KUKA KRL data list: ps_a_etb_res_c02.dat

&ACCESS RVO1
&REL 341
&COMMENT Solda Atego ETB
&PARAM DISKPATH = KRC:\R1\Program\OLP
DEFDAT  ps_a_etb_res_c02
;FOLD EXTERNAL DECLARATIONS;%{PE}%MKUKATPBASIS,%CEXT,%VCOMMON,%P
;FOLD GRIPPERTECH EXT
EXT  H50 (INT  :IN,INT  :IN,INT  :IN,GRP_TYP  :IN )
;ENDFOLD (GRIPPERTECH EXT)
;FOLD SPOTTECH EXT
EXT  USERSPOT (S_COMMAND  :IN,SPOT_TYPE  :IN )
;ENDFOLD (SPOTTECH EXT)
;FOLD BASISTECH EXT;%{PE}%MKUKATPBASIS,%CEXT,%VEXT,%P
EXT  BAS (BAS_COMMAND  :IN,REAL  :IN )
DECL INT SUCCESS
;ENDFOLD (BASISTECH EXT)
;FOLD USER EXT;%{E}%MKUKATPUSER,%CEXT,%VEXT,%P
;Make your modifications here

;ENDFOLD (USER EXT)
;ENDFOLD (EXTERNAL DECLARATIONS)
DECL FDAT Fl015={TOOL_NO 3,BASE_NO 3,IPO_FRAME #BASE,POINT2[] " "}
DECL E6POS Xl015={X 31.0238705,Y -594.734375,Z 749.761108,A -124.005302,B 73.4685669,C -126.8536,S 18,T 35,E1 0.0,E2 0.0,E3 0.0,E4 0.0,E5 0.0,E6 0.0}
DECL LDAT LL_OLP3={VEL 2.0,ACC 100.0,APO_DIST 0.0,APO_FAC 0.0,ORI_TYP #VAR,CIRC_TYP #BASE,JERK_FAC 50.0}
DECL FDAT Fl020={TOOL_NO 3,BASE_NO 3,IPO_FRAME #BASE,POINT2[] " "}
DECL E6POS Xl020={X 52.5596504,Y -663.980286,Z 782.928284,A -123.990501,B 73.4740219,C -126.844803,S 18,T 35,E1 0.0,E2 0.0,E3 0.0,E4 0.0,E5 0.0,E6 0.0}
DECL LDAT LL_OLP4={VEL 2.0,ACC 100.0,APO_DIST 150.0,APO_FAC 0.0,ORI_TYP #VAR,CIRC_TYP #BASE,JERK_FAC 50.0}
DECL FDAT Fl025={TOOL_NO 3,BASE_NO 3,IPO_FRAME #BASE,POINT2[] " "}
DECL E6POS Xl025={X 114.589798,Y -708.233398,Z 735.784912,A -94.4452896,B 74.9285278,C -94.8186569,S 18,T 35,E1 0.0,E2 0.0,E3 0.0,E4 0.0,E5 0.0,E6 0.0}
DECL LDAT LL_OLP5={VEL 2.0,ACC 100.0,APO_DIST 150.0,APO_FAC 0.0,ORI_TYP #VAR,CIRC_TYP #BASE,JERK_FAC 50.0}
DECL FDAT Fl030={TOOL_NO 3,BASE_NO 3,IPO_FRAME #BASE,POINT2[] " "}
DECL E6POS Xl030={X 274.340912,Y -703.442017,Z 641.453125,A -54.7125397,B 69.4866562,C -51.1110687,S 18,T 35,E1 0.0,E2 0.0,E3 0.0,E4 0.0,E5 0.0,E6 0.0}
DECL LDAT LL_OLP6={VEL 2.0,ACC 100.0,APO_DIST 150.0,APO_FAC 0.0,ORI_TYP #VAR,CIRC_TYP #BASE,JERK_FAC 50.0}
DECL FDAT Fl035={TOOL_NO 3,BASE_NO 3,IPO_FRAME #BASE,POINT2[] " "}
DECL E6POS Xl035={X 587.583008,Y -653.065002,Z 418.535004,A -24.4300995,B 45.0119019,C -12.2528,S 2,T 35}
DECL LDAT LL_OLP7={VEL 2.0,ACC 100.0,APO_DIST 150.0,APO_FAC 0.0,ORI_TYP #VAR,CIRC_TYP #BASE,JERK_FAC 50.0}
DECL FDAT Fl040={TOOL_NO 3,BASE_NO 3,IPO_FRAME #BASE,POINT2[] " "}
DECL E6POS Xl040={X 713.926392,Y -668.47052,Z 338.3591,A -21.6110992,B 32.5932884,C -7.47571993,S 18,T 35,E1 0.0,E2 0.0,E3 0.0,E4 0.0,E5 0.0,E6 0.0}
DECL LDAT LL_OLP8={VEL 2.0,ACC 100.0,APO_DIST 150.0,APO_FAC 0.0,ORI_TYP #VAR,CIRC_TYP #BASE,JERK_FAC 50.0}
DECL FDAT Fl045={TOOL_NO 3,BASE_NO 3,IPO_FRAME #BASE,POINT2[] " "}
DECL E6POS Xl045={X 765.193115,Y -1115.46997,Z 133.110596,A -16.9657192,B 14.9491901,C -20.2578106,S 18,T 3,E1 0.0,E2 0.0,E3 0.0,E4 0.0,E5 0.0,E6 0.0}
DECL LDAT LL_OLP9={VEL 2.0,ACC 100.0,APO_DIST 150.0,APO_FAC 0.0,ORI_TYP #VAR,CIRC_TYP #BASE,JERK_FAC 50.0}
DECL FDAT Fl050={TOOL_NO 3,BASE_NO 3,IPO_FRAME #BASE,POINT2[] " "}
DECL E6POS Xl050={X 746.955017,Y -2151.34399,Z 121.584,A -16.3197002,B 12.0216999,C -22.6774998,S 2,T 3}
DECL FDAT Fl055={TOOL_NO 3,BASE_NO 3,IPO_FRAME #BASE,POINT2[] " "}
DECL E6POS Xl055={X 1024.95605,Y -2151.34399,Z 535.583008,A 28.6604996,B 24.3521996,C -7.86679983,S 2,T 3}
DECL FDAT Fl060={TOOL_NO 3,BASE_NO 3,IPO_FRAME #BASE,POINT2[] " "}
DECL PDAT PP_OLP2={VEL 100.0,ACC 100.0,APO_DIST 100.0,APO_MODE #CDIS}
DECL E6POS Xl060={X 1158.77795,Y -1627.54797,Z 929.039001,A 43.2759018,B -40.0696983,C 26.0069008,S 6,T 19}
DECL FDAT Fl065={TOOL_NO 3,BASE_NO 3,IPO_FRAME #BASE,POINT2[] " "}
DECL PDAT PP_OLP3={VEL 100.0,ACC 100.0,APO_DIST 30.0,APO_MODE #CDIS}
DECL E6POS Xl065={X 868.09668,Y -1244.59497,Z 1101.58606,A 29.2385902,B -63.5374794,C 57.4689713,S 22,T 19,E1 0.0,E2 0.0,E3 0.0,E4 0.0,E5 0.0,E6 0.0}
DECL FDAT Fl070={TOOL_NO 3,BASE_NO 3,IPO_FRAME #BASE,POINT2[] " "}
DECL PDAT PP_OLP4={VEL 100.0,ACC 100.0,APO_DIST 30.0,APO_MODE #CDIS}
DECL E6POS Xl070={X 814.102905,Y -929.709717,Z 1165.05896,A 29.5652695,B -64.2360001,C 60.087719,S 22,T 19,E1 0.0,E2 0.0,E3 0.0,E4 0.0,E5 0.0,E6 0.0}
DECL E6POS XSWP_60_7787={X 556.251099,Y -975.593323,Z 1302.83704,A 143.936295,B -83.3156891,C -51.7027016,S 18,T 43,E1 0.0,E2 0.0,E3 0.0,E4 0.0,E5 0.0,E6 0.0}
DECL FDAT FSWP_60_7787={TOOL_NO 3,BASE_NO 3,IPO_FRAME #BASE,POINT2[] " "}
DECL LDAT LL_OLP12={VEL 2.0,ACC 100.0,APO_DIST 0.0,APO_FAC 0.0,ORI_TYP #VAR,CIRC_TYP #BASE,JERK_FAC 50.0}
DECL E6POS XSWP_60_7789={X 584.018677,Y -975.191223,Z 1304.28101,A 144.007706,B -83.3220673,C -54.6376801,S 18,T 43,E1 0.0,E2 0.0,E3 0.0,E4 0.0,E5 0.0,E6 0.0}
DECL FDAT FSWP_60_7789={TOOL_NO 3,BASE_NO 3,IPO_FRAME #BASE,POINT2[] " "}
DECL LDAT LL_OLP13={VEL 2.0,ACC 100.0,APO_DIST 0.0,APO_FAC 0.0,ORI_TYP #VAR,CIRC_TYP #BASE,JERK_FAC 50.0}
DECL E6POS XSWP_60_7791={X 613.247986,Y -978.535706,Z 1306.79395,A 144.016205,B -83.3237762,C -54.6469498,S 22,T 19,E1 0.0,E2 0.0,E3 0.0,E4 0.0,E5 0.0,E6 0.0}
DECL FDAT FSWP_60_7791={TOOL_NO 3,BASE_NO 3,IPO_FRAME #BASE,POINT2[] " "}
DECL LDAT LL_OLP14={VEL 2.0,ACC 100.0,APO_DIST 0.0,APO_FAC 0.0,ORI_TYP #VAR,CIRC_TYP #BASE,JERK_FAC 50.0}
DECL FDAT Fl075={TOOL_NO 3,BASE_NO 3,IPO_FRAME #BASE,POINT2[] " "}
DECL E6POS Xl075={X 647.49408,Y -968.108398,Z 1301.578,A 26.10993,B -81.5293198,C 62.8230019,S 22,T 19,E1 0.0,E2 0.0,E3 0.0,E4 0.0,E5 0.0,E6 0.0}
DECL LDAT LL_OLP15={VEL 2.0,ACC 100.0,APO_DIST 10.0,APO_FAC 0.0,ORI_TYP #VAR,CIRC_TYP #BASE,JERK_FAC 50.0}
DECL E6POS XSWP_60_7795={X 702.531372,Y -979.488403,Z 1310.90405,A 26.1140499,B -81.5290985,C 62.8173103,S 22,T 19,E1 0.0,E2 0.0,E3 0.0,E4 0.0,E5 0.0,E6 0.0}
DECL FDAT FSWP_60_7795={TOOL_NO 3,BASE_NO 3,IPO_FRAME #BASE,POINT2[] " "}
DECL LDAT LL_OLP16={VEL 2.0,ACC 100.0,APO_DIST 0.0,APO_FAC 0.0,ORI_TYP #VAR,CIRC_TYP #BASE,JERK_FAC 50.0}
DECL E6POS XSWP_60_7797={X 744.206726,Y -979.352295,Z 1312.43701,A 26.1139603,B -81.5292435,C 62.8172798,S 22,T 19,E1 0.0,E2 0.0,E3 0.0,E4 0.0,E5 0.0,E6 0.0}
DECL FDAT FSWP_60_7797={TOOL_NO 3,BASE_NO 3,IPO_FRAME #BASE,POINT2[] " "}
DECL LDAT LL_OLP17={VEL 2.0,ACC 100.0,APO_DIST 0.0,APO_FAC 0.0,ORI_TYP #VAR,CIRC_TYP #BASE,JERK_FAC 50.0}
DECL E6POS XSWP_60_7799={X 790.615112,Y -980.393005,Z 1313.89502,A 26.1141491,B -81.5294495,C 62.8168793,S 22,T 19,E1 0.0,E2 0.0,E3 0.0,E4 0.0,E5 0.0,E6 0.0}
DECL FDAT FSWP_60_7799={TOOL_NO 3,BASE_NO 3,IPO_FRAME #BASE,POINT2[] " "}
DECL LDAT LL_OLP18={VEL 2.0,ACC 100.0,APO_DIST 0.0,APO_FAC 0.0,ORI_TYP #VAR,CIRC_TYP #BASE,JERK_FAC 50.0}
DECL E6POS XSWP_60_7801={X 838.112976,Y -981.874023,Z 1316.401,A 26.1212902,B -81.5292511,C 62.8090897,S 22,T 19,E1 0.0,E2 0.0,E3 0.0,E4 0.0,E5 0.0,E6 0.0}
DECL FDAT FSWP_60_7801={TOOL_NO 3,BASE_NO 3,IPO_FRAME #BASE,POINT2[] " "}
DECL LDAT LL_OLP19={VEL 2.0,ACC 100.0,APO_DIST 0.0,APO_FAC 0.0,ORI_TYP #VAR,CIRC_TYP #BASE,JERK_FAC 50.0}
DECL E6POS XSWP_60_7803={X 879.085815,Y -982.434204,Z 1317.19104,A 26.1254692,B -81.5289612,C 62.8045807,S 22,T 19,E1 0.0,E2 0.0,E3 0.0,E4 0.0,E5 0.0,E6 0.0}
DECL FDAT FSWP_60_7803={TOOL_NO 3,BASE_NO 3,IPO_FRAME #BASE,POINT2[] " "}
DECL LDAT LL_OLP20={VEL 2.0,ACC 100.0,APO_DIST 0.0,APO_FAC 0.0,ORI_TYP #VAR,CIRC_TYP #BASE,JERK_FAC 50.0}
DECL E6POS XSWP_60_7807={X 972.588501,Y -983.796387,Z 1320.14001,A 26.1272507,B -81.5321884,C 62.805069,S 22,T 19,E1 0.0,E2 0.0,E3 0.0,E4 0.0,E5 0.0,E6 0.0}
DECL FDAT FSWP_60_7807={TOOL_NO 3,BASE_NO 3,IPO_FRAME #BASE,POINT2[] " "}
DECL LDAT LL_OLP21={VEL 2.0,ACC 100.0,APO_DIST 0.0,APO_FAC 0.0,ORI_TYP #VAR,CIRC_TYP #BASE,JERK_FAC 50.0}
DECL E6POS XSWP_60_7809={X 1019.99597,Y -984.109985,Z 1320.86499,A 26.1021805,B -81.5284271,C 62.8301506,S 22,T 19,E1 0.0,E2 0.0,E3 0.0,E4 0.0,E5 0.0,E6 0.0}
DECL FDAT FSWP_60_7809={TOOL_NO 3,BASE_NO 3,IPO_FRAME #BASE,POINT2[] " "}
DECL LDAT LL_OLP22={VEL 2.0,ACC 100.0,APO_DIST 0.0,APO_FAC 0.0,ORI_TYP #VAR,CIRC_TYP #BASE,JERK_FAC 50.0}
DECL E6POS XSWP_60_7811={X 1062.02405,Y -985.307312,Z 1321.88196,A 26.1204891,B -81.530159,C 62.8099213,S 22,T 19,E1 0.0,E2 0.0,E3 0.0,E4 0.0,E5 0.0,E6 0.0}
DECL FDAT FSWP_60_7811={TOOL_NO 3,BASE_NO 3,IPO_FRAME #BASE,POINT2[] " "}
DECL LDAT LL_OLP23={VEL 2.0,ACC 100.0,APO_DIST 0.0,APO_FAC 0.0,ORI_TYP #VAR,CIRC_TYP #BASE,JERK_FAC 50.0}
DECL E6POS XSWP_60_7813={X 1102.52795,Y -985.327515,Z 1323.27405,A 26.1103802,B -81.5287933,C 62.8201218,S 22,T 19,E1 0.0,E2 0.0,E3 0.0,E4 0.0,E5 0.0,E6 0.0}
DECL FDAT FSWP_60_7813={TOOL_NO 3,BASE_NO 3,IPO_FRAME #BASE,POINT2[] " "}
DECL LDAT LL_OLP24={VEL 2.0,ACC 100.0,APO_DIST 0.0,APO_FAC 0.0,ORI_TYP #VAR,CIRC_TYP #BASE,JERK_FAC 50.0}
DECL E6POS XSWP_60_7815={X 1147.90198,Y -985.572815,Z 1324.37402,A 26.1104202,B -81.528923,C 62.8199615,S 22,T 19,E1 0.0,E2 0.0,E3 0.0,E4 0.0,E5 0.0,E6 0.0}
DECL FDAT FSWP_60_7815={TOOL_NO 3,BASE_NO 3,IPO_FRAME #BASE,POINT2[] " "}
DECL LDAT LL_OLP25={VEL 2.0,ACC 100.0,APO_DIST 0.0,APO_FAC 0.0,ORI_TYP #VAR,CIRC_TYP #BASE,JERK_FAC 50.0}
DECL FDAT Fl080={TOOL_NO 3,BASE_NO 3,IPO_FRAME #BASE,POINT2[] " "}
DECL E6POS Xl080={X 1163.40503,Y -974.013977,Z 1320.32605,A 13.9886799,B -81.9076538,C 74.8192825,S 22,T 19,E1 0.0,E2 0.0,E3 0.0,E4 0.0,E5 0.0,E6 0.0}
DECL LDAT LL_OLP26={VEL 2.0,ACC 100.0,APO_DIST 150.0,APO_FAC 0.0,ORI_TYP #VAR,CIRC_TYP #BASE,JERK_FAC 50.0}
DECL FDAT Fl085={TOOL_NO 3,BASE_NO 3,IPO_FRAME #BASE,POINT2[] " "}
DECL E6POS Xl085={X 1163.94604,Y -969.89032,Z 1259.79297,A 17.7539597,B -81.8335037,C 71.0904465,S 22,T 19,E1 0.0,E2 0.0,E3 0.0,E4 0.0,E5 0.0,E6 0.0}
DECL LDAT LL_OLP27={VEL 2.0,ACC 100.0,APO_DIST 150.0,APO_FAC 0.0,ORI_TYP #VAR,CIRC_TYP #BASE,JERK_FAC 50.0}
DECL FDAT Fl090={TOOL_NO 3,BASE_NO 3,IPO_FRAME #BASE,POINT2[] " "}
DECL E6POS Xl090={X 983.369995,Y -1478.85596,Z 590.278015,A 179.957108,B -45.9999008,C -90.0,S 6,T 19}
DECL LDAT LL_OLP28={VEL 2.0,ACC 100.0,APO_DIST 150.0,APO_FAC 0.0,ORI_TYP #VAR,CIRC_TYP #BASE,JERK_FAC 50.0}
DECL FDAT Fl100={TOOL_NO 3,BASE_NO 3,IPO_FRAME #BASE,POINT2[] " "}
DECL E6POS Xl100={X 1306.58801,Y -1016.62402,Z 103.935699,A 179.322601,B -25.2803707,C -90.9719391,S 22,T 19,E1 0.0,E2 0.0,E3 0.0,E4 0.0,E5 0.0,E6 0.0}
DECL LDAT LL_OLP30={VEL 2.0,ACC 100.0,APO_DIST 0.0,APO_FAC 0.0,ORI_TYP #VAR,CIRC_TYP #BASE,JERK_FAC 50.0}
DECL FDAT FSWP_60_7487={TOOL_NO 3,BASE_NO 3,IPO_FRAME #BASE,POINT2[] " "}
DECL E6POS XSWP_60_7487={X 1306.44397,Y -1021.547,Z 118.262802,A 179.322403,B -25.28022,C -90.9719391,S 18,T 43,E1 0.0,E2 0.0,E3 0.0,E4 0.0,E5 0.0,E6 0.0}
DECL LDAT LL_OLP31={VEL 2.0,ACC 100.0,APO_DIST 0.0,APO_FAC 0.0,ORI_TYP #VAR,CIRC_TYP #BASE,JERK_FAC 50.0}
DECL FDAT FSWP_60_7489={TOOL_NO 3,BASE_NO 3,IPO_FRAME #BASE,POINT2[] " "}
DECL E6POS XSWP_60_7489={X 1339.98206,Y -1023.56598,Z 120.081001,A 179.952698,B -20.9994793,C -93.3431702,S 18,T 43,E1 0.0,E2 0.0,E3 0.0,E4 0.0,E5 0.0,E6 0.0}
DECL LDAT LL_OLP32={VEL 2.0,ACC 100.0,APO_DIST 0.0,APO_FAC 0.0,ORI_TYP #VAR,CIRC_TYP #BASE,JERK_FAC 50.0}
DECL FDAT FSWP_60_7491={TOOL_NO 3,BASE_NO 3,IPO_FRAME #BASE,POINT2[] " "}
DECL E6POS XSWP_60_7491={X 1370.55298,Y -1021.91803,Z 121.484901,A -179.790604,B -20.8528404,C -93.2146988,S 18,T 43,E1 0.0,E2 0.0,E3 0.0,E4 0.0,E5 0.0,E6 0.0}
DECL LDAT LL_OLP33={VEL 2.0,ACC 100.0,APO_DIST 0.0,APO_FAC 0.0,ORI_TYP #VAR,CIRC_TYP #BASE,JERK_FAC 50.0}
DECL FDAT Fl105={TOOL_NO 3,BASE_NO 3,IPO_FRAME #BASE,POINT2[] " "}
DECL E6POS Xl105={X 1373.94495,Y -1013.10602,Z 88.1965637,A 179.956894,B -18.0000401,C -89.9994507,S 22,T 19,E1 0.0,E2 0.0,E3 0.0,E4 0.0,E5 0.0,E6 0.0}
DECL LDAT LL_OLP34={VEL 2.0,ACC 100.0,APO_DIST 0.0,APO_FAC 0.0,ORI_TYP #VAR,CIRC_TYP #BASE,JERK_FAC 50.0}
DECL FDAT Fl110={TOOL_NO 3,BASE_NO 3,IPO_FRAME #BASE,POINT2[] " "}
DECL E6POS Xl110={X 1469.69604,Y -999.753174,Z 86.6159668,A 179.956894,B -19.0000801,C -89.9993668,S 22,T 19,E1 0.0,E2 0.0,E3 0.0,E4 0.0,E5 0.0,E6 0.0}
DECL LDAT LL_OLP35={VEL 2.0,ACC 100.0,APO_DIST 0.0,APO_FAC 0.0,ORI_TYP #VAR,CIRC_TYP #BASE,JERK_FAC 50.0}
DECL FDAT FSWP_60_7495={TOOL_NO 3,BASE_NO 3,IPO_FRAME #BASE,POINT2[] " "}
DECL E6POS XSWP_60_7495={X 1442.27197,Y -1019.48102,Z 122.377296,A 179.957199,B -20.9995899,C -93.1918564,S 22,T 19,E1 0.0,E2 0.0,E3 0.0,E4 0.0,E5 0.0,E6 0.0}
DECL LDAT LL_OLP36={VEL 2.0,ACC 100.0,APO_DIST 0.0,APO_FAC 0.0,ORI_TYP #VAR,CIRC_TYP #BASE,JERK_FAC 50.0}
DECL FDAT FSWP_60_7497={TOOL_NO 3,BASE_NO 3,IPO_FRAME #BASE,POINT2[] " "}
DECL E6POS XSWP_60_7497={X 1479.71106,Y -1018.96399,Z 124.096703,A -179.6689,B -20.9927502,C -93.8000717,S 18,T 43,E1 0.0,E2 0.0,E3 0.0,E4 0.0,E5 0.0,E6 0.0}
DECL LDAT LL_OLP37={VEL 2.0,ACC 100.0,APO_DIST 0.0,APO_FAC 0.0,ORI_TYP #VAR,CIRC_TYP #BASE,JERK_FAC 50.0}
DECL FDAT FSWP_60_7499={TOOL_NO 3,BASE_NO 3,IPO_FRAME #BASE,POINT2[] " "}
DECL E6POS XSWP_60_7499={X 1519.71802,Y -1018.96802,Z 124.852798,A -179.660904,B -20.9865093,C -93.8057938,S 18,T 43,E1 0.0,E2 0.0,E3 0.0,E4 0.0,E5 0.0,E6 0.0}
DECL LDAT LL_OLP38={VEL 2.0,ACC 100.0,APO_DIST 0.0,APO_FAC 0.0,ORI_TYP #VAR,CIRC_TYP #BASE,JERK_FAC 50.0}
DECL FDAT Fl115={TOOL_NO 3,BASE_NO 3,IPO_FRAME #BASE,POINT2[] " "}
DECL E6POS Xl115={X 1563.23596,Y -1006.01099,Z 70.940239,A 179.949402,B -20.9986,C -89.9980469,S 22,T 19,E1 0.0,E2 0.0,E3 0.0,E4 0.0,E5 0.0,E6 0.0}
DECL LDAT LL_OLP39={VEL 2.0,ACC 100.0,APO_DIST 150.0,APO_FAC 0.0,ORI_TYP #VAR,CIRC_TYP #BASE,JERK_FAC 50.0}
DECL FDAT Fl120={TOOL_NO 3,BASE_NO 3,IPO_FRAME #BASE,POINT2[] " "}
DECL E6POS Xl120={X 1563.09998,Y -1231.07898,Z 75.473999,A 179.957108,B -20.9999008,C -90.0,S 6,T 19}
DECL LDAT LL_OLP40={VEL 2.0,ACC 100.0,APO_DIST 150.0,APO_FAC 0.0,ORI_TYP #VAR,CIRC_TYP #BASE,JERK_FAC 50.0}
DECL FDAT Fl125={TOOL_NO 3,BASE_NO 3,IPO_FRAME #BASE,POINT2[] " "}
DECL E6POS Xl125={X 1667.94995,Y -1726.27698,Z 177.965393,A 179.960098,B -45.9984512,C -90.0082397,S 22,T 19,E1 0.0,E2 0.0,E3 0.0,E4 0.0,E5 0.0,E6 0.0}
DECL BASIS_SUGG_T LAST_BASIS={POINT1[] "P16                     ",POINT2[] "P16                     ",CP_PARAMS[] "CPDAT0                  ",PTP_PARAMS[] "PDAT17                  ",CONT[] "C_DIS                   ",CP_VEL[] "2                       ",PTP_VEL[] "100                     ",SYNC_PARAMS[] "SYNCDAT                 ",SPL_NAME[] "S0                      "}
DECL PDAT PP_OLP6={VEL 100.0,ACC 100.0,APO_DIST 0.0}
DECL E6POS Xl006={X 746.955017,Y -2151.34399,Z 121.584,A -16.3197002,B 12.0216999,C -22.6774998,S 2,T 3}
DECL FDAT Fl006={TOOL_NO 3,BASE_NO 3,IPO_FRAME #BASE,POINT2[] " "}
DECL LDAT LL_OLP42={VEL 2.0,ACC 100.0,APO_DIST 30.0,APO_FAC 0.0,ORI_TYP #VAR,CIRC_TYP #BASE,JERK_FAC 50.0}
DECL E6POS Xl011={X 745.054077,Y -1210.42102,Z 45.7849503,A -16.3183804,B 12.0204601,C -22.6786194,S 18,T 3,E1 0.0,E2 0.0,E3 0.0,E4 0.0,E5 0.0,E6 0.0}
DECL FDAT Fl011={TOOL_NO 3,BASE_NO 3,IPO_FRAME #BASE,POINT2[] " "}
DECL E6POS Xl016={X 960.239685,Y -695.417419,Z 224.849792,A -18.2002106,B 11.2452402,C -1.07748699,S 18,T 3,E1 0.0,E2 0.0,E3 0.0,E4 0.0,E5 0.0,E6 0.0}
DECL FDAT Fl016={TOOL_NO 3,BASE_NO 3,IPO_FRAME #BASE,POINT2[] " "}
DECL LDAT LL_OLP44={VEL 2.0,ACC 100.0,APO_DIST 10.0,APO_FAC 0.0,ORI_TYP #VAR,CIRC_TYP #BASE,JERK_FAC 50.0}
DECL E6POS Xl021={X 587.583008,Y -653.065002,Z 418.535004,A -24.4300995,B 45.0119019,C -12.2528,S 2,T 35}
DECL FDAT Fl021={TOOL_NO 3,BASE_NO 3,IPO_FRAME #BASE,POINT2[] " "}
DECL LDAT LL_OLP45={VEL 2.0,ACC 100.0,APO_DIST 10.0,APO_FAC 0.0,ORI_TYP #VAR,CIRC_TYP #BASE,JERK_FAC 50.0}
DECL E6POS Xl026={X 343.014008,Y -642.028076,Z 721.553772,A -44.0348091,B 69.0998383,C -36.2288399,S 18,T 35,E1 0.0,E2 0.0,E3 0.0,E4 0.0,E5 0.0,E6 0.0}
DECL FDAT Fl026={TOOL_NO 3,BASE_NO 3,IPO_FRAME #BASE,POINT2[] " "}
DECL LDAT LL_OLP46={VEL 2.0,ACC 100.0,APO_DIST 10.0,APO_FAC 0.0,ORI_TYP #VAR,CIRC_TYP #BASE,JERK_FAC 50.0}
DECL E6POS Xl031={X 328.106598,Y -647.627686,Z 744.279175,A -69.6208572,B 74.6609573,C -62.4694595,S 18,T 35,E1 0.0,E2 0.0,E3 0.0,E4 0.0,E5 0.0,E6 0.0}
DECL FDAT Fl031={TOOL_NO 3,BASE_NO 3,IPO_FRAME #BASE,POINT2[] " "}
DECL LDAT LL_OLP47={VEL 2.0,ACC 100.0,APO_DIST 10.0,APO_FAC 0.0,ORI_TYP #VAR,CIRC_TYP #BASE,JERK_FAC 50.0}
DECL E6POS Xl036={X 129.093597,Y -809.958801,Z 712.43811,A -122.0411,B 73.8237534,C -124.462097,S 18,T 35,E1 0.0,E2 0.0,E3 0.0,E4 0.0,E5 0.0,E6 0.0}
DECL FDAT Fl036={TOOL_NO 3,BASE_NO 3,IPO_FRAME #BASE,POINT2[] " "}
DECL LDAT LL_OLP48={VEL 2.0,ACC 100.0,APO_DIST 10.0,APO_FAC 0.0,ORI_TYP #VAR,CIRC_TYP #BASE,JERK_FAC 50.0}
DECL E6POS Xl041={X 111.864998,Y -869.716003,Z 602.434021,A -124.114799,B 73.5134964,C -126.966202,S 2,T 35}
DECL FDAT Fl041={TOOL_NO 3,BASE_NO 3,IPO_FRAME #BASE,POINT2[] " "}
DECL LDAT LL_OLP49={VEL 2.0,ACC 100.0,APO_DIST 0.0,APO_FAC 0.0,ORI_TYP #VAR,CIRC_TYP #BASE,JERK_FAC 50.0}
DECL E6POS XSWP_60_7909={X 133.370605,Y -867.391907,Z 600.803284,A -109.557999,B 75.6781464,C -117.705002,S 18,T 35,E1 0.0,E2 0.0,E3 0.0,E4 0.0,E5 0.0,E6 0.0}
DECL FDAT FSWP_60_7909={TOOL_NO 3,BASE_NO 3,IPO_FRAME #BASE,POINT2[] " "}
DECL E6POS XSWP_60_7907={X 129.188995,Y -831.960022,Z 602.795776,A -109.579597,B 75.6635437,C -112.607803,S 18,T 35,E1 0.0,E2 0.0,E3 0.0,E4 0.0,E5 0.0,E6 0.0}
DECL FDAT FSWP_60_7907={TOOL_NO 3,BASE_NO 3,IPO_FRAME #BASE,POINT2[] " ",TQ_STATE FALSE}
DECL LDAT LL_OLP51={VEL 2.0,ACC 100.0,APO_DIST 0.0,APO_FAC 0.0,ORI_TYP #VAR,CIRC_TYP #BASE,JERK_FAC 50.0}
DECL E6POS XSWP_60_7905={X 118.431503,Y -758.19519,Z 600.044189,A -94.7613678,B 76.664772,C -98.2709122,S 18,T 35,E1 0.0,E2 0.0,E3 0.0,E4 0.0,E5 0.0,E6 0.0}
DECL FDAT FSWP_60_7905={TOOL_NO 3,BASE_NO 3,IPO_FRAME #BASE,POINT2[] " "}
DECL LDAT LL_OLP52={VEL 2.0,ACC 100.0,APO_DIST 0.0,APO_FAC 0.0,ORI_TYP #VAR,CIRC_TYP #BASE,JERK_FAC 50.0}
DECL E6POS XSWP_60_7903={X 114.063904,Y -728.930908,Z 599.57019,A -101.589203,B 80.7481232,C -104.514198,S 18,T 35,E1 0.0,E2 0.0,E3 0.0,E4 0.0,E5 0.0,E6 0.0}
DECL FDAT FSWP_60_7903={TOOL_NO 3,BASE_NO 3,IPO_FRAME #BASE,POINT2[] " "}
DECL LDAT LL_OLP53={VEL 2.0,ACC 100.0,APO_DIST 0.0,APO_FAC 0.0,ORI_TYP #VAR,CIRC_TYP #BASE,JERK_FAC 50.0}
DECL E6POS XSWP_60_7901={X 112.070602,Y -698.476318,Z 599.263123,A -103.006798,B 80.6964798,C -105.953697,S 18,T 35,E1 0.0,E2 0.0,E3 0.0,E4 0.0,E5 0.0,E6 0.0}
DECL FDAT FSWP_60_7901={TOOL_NO 3,BASE_NO 3,IPO_FRAME #BASE,POINT2[] " "}
DECL LDAT LL_OLP54={VEL 2.0,ACC 100.0,APO_DIST 0.0,APO_FAC 0.0,ORI_TYP #VAR,CIRC_TYP #BASE,JERK_FAC 50.0}
DECL E6POS XSWP_60_7329={X 100.614502,Y -668.871277,Z 599.434021,A -105.788803,B 80.5839996,C -108.767899,S 18,T 35,E1 0.0,E2 0.0,E3 0.0,E4 0.0,E5 0.0,E6 0.0}
DECL FDAT FSWP_60_7329={TOOL_NO 3,BASE_NO 3,IPO_FRAME #BASE,POINT2[] " "}
DECL LDAT LL_OLP55={VEL 2.0,ACC 100.0,APO_DIST 0.0,APO_FAC 0.0,ORI_TYP #VAR,CIRC_TYP #BASE,JERK_FAC 50.0}
DECL E6POS XSWP_60_7893={X 98.5761185,Y -581.989014,Z 599.465881,A -106.232101,B 80.5538635,C -106.072998,S 18,T 35,E1 0.0,E2 0.0,E3 0.0,E4 0.0,E5 0.0,E6 0.0}
DECL FDAT FSWP_60_7893={TOOL_NO 3,BASE_NO 3,IPO_FRAME #BASE,POINT2[] " "}
DECL LDAT LL_OLP56={VEL 2.0,ACC 100.0,APO_DIST 0.0,APO_FAC 0.0,ORI_TYP #VAR,CIRC_TYP #BASE,JERK_FAC 50.0}
DECL E6POS XSWP_60_7891={X 101.4776,Y -547.356323,Z 601.088318,A -147.087204,B 85.1514587,C -145.4216,S 18,T 35,E1 0.0,E2 0.0,E3 0.0,E4 0.0,E5 0.0,E6 0.0}
DECL FDAT FSWP_60_7891={TOOL_NO 3,BASE_NO 3,IPO_FRAME #BASE,POINT2[] " "}
DECL LDAT LL_OLP57={VEL 2.0,ACC 100.0,APO_DIST 0.0,APO_FAC 0.0,ORI_TYP #VAR,CIRC_TYP #BASE,JERK_FAC 50.0}
DECL E6POS XSWP_60_7889={X 91.583313,Y -514.910889,Z 602.981873,A -155.413101,B 84.5177765,C -154.862106,S 18,T 35,E1 0.0,E2 0.0,E3 0.0,E4 0.0,E5 0.0,E6 0.0}
DECL FDAT FSWP_60_7889={TOOL_NO 3,BASE_NO 3,IPO_FRAME #BASE,POINT2[] " "}
DECL LDAT LL_OLP58={VEL 2.0,ACC 100.0,APO_DIST 0.0,APO_FAC 0.0,ORI_TYP #VAR,CIRC_TYP #BASE,JERK_FAC 50.0}
DECL E6POS XSWP_60_7887={X 84.9992828,Y -481.50061,Z 603.889771,A -106.016602,B 71.1151123,C -109.612396,S 18,T 35,E1 0.0,E2 0.0,E3 0.0,E4 0.0,E5 0.0,E6 0.0}
DECL FDAT FSWP_60_7887={TOOL_NO 3,BASE_NO 3,IPO_FRAME #BASE,POINT2[] " "}
DECL LDAT LL_OLP59={VEL 2.0,ACC 100.0,APO_DIST 0.0,APO_FAC 0.0,ORI_TYP #VAR,CIRC_TYP #BASE,JERK_FAC 50.0}
DECL E6POS XSWP_60_7885={X 97.2219772,Y -448.786713,Z 600.723206,A -109.852203,B 72.9984512,C -112.345001,S 18,T 35,E1 0.0,E2 0.0,E3 0.0,E4 0.0,E5 0.0,E6 0.0}
DECL FDAT FSWP_60_7885={TOOL_NO 3,BASE_NO 3,IPO_FRAME #BASE,POINT2[] " "}
DECL LDAT LL_OLP60={VEL 2.0,ACC 100.0,APO_DIST 0.0,APO_FAC 0.0,ORI_TYP #VAR,CIRC_TYP #BASE,JERK_FAC 50.0}
DECL E6POS XSWP_60_7883={X 95.7474594,Y -416.565308,Z 601.213013,A -113.249001,B 74.3331528,C -114.915604,S 18,T 35,E1 0.0,E2 0.0,E3 0.0,E4 0.0,E5 0.0,E6 0.0}
DECL FDAT FSWP_60_7883={TOOL_NO 3,BASE_NO 3,IPO_FRAME #BASE,POINT2[] " "}
DECL LDAT LL_OLP61={VEL 2.0,ACC 100.0,APO_DIST 0.0,APO_FAC 0.0,ORI_TYP #VAR,CIRC_TYP #BASE,JERK_FAC 50.0}
DECL E6POS XSWP_60_7881={X 93.8382721,Y -383.756592,Z 600.205017,A -121.905899,B 78.0305862,C -124.633202,S 18,T 35,E1 0.0,E2 0.0,E3 0.0,E4 0.0,E5 0.0,E6 0.0}
DECL FDAT FSWP_60_7881={TOOL_NO 3,BASE_NO 3,IPO_FRAME #BASE,POINT2[] " "}
DECL LDAT LL_OLP62={VEL 2.0,ACC 100.0,APO_DIST 150.0,APO_FAC 0.0,ORI_TYP #VAR,CIRC_TYP #BASE,JERK_FAC 50.0}
DECL E6POS Xl046={X 97.8552628,Y -435.905701,Z 624.627991,A -119.415398,B 74.1074066,C -123.265099,S 18,T 35,E1 0.0,E2 0.0,E3 0.0,E4 0.0,E5 0.0,E6 0.0}
DECL FDAT Fl046={TOOL_NO 3,BASE_NO 3,IPO_FRAME #BASE,POINT2[] " "}
DECL LDAT LCPDAT1={VEL 2.0,ACC 100.0,APO_DIST 100.0,APO_FAC 50.0,AXIS_VEL 100.0,AXIS_ACC 100.0,ORI_TYP #VAR,CIRC_TYP #BASE,JERK_FAC 50.0,GEAR_JERK 50.0,EXAX_IGN 0}
DECL E6POS XP4={X 54.6556282,Y -541.398315,Z 612.695313,A -158.196899,B 83.6885376,C -157.655106,S 18,T 35,E1 0.0,E2 0.0,E3 0.0,E4 0.0,E5 0.0,E6 0.0}
DECL FDAT FP4={TOOL_NO 3,BASE_NO 3,IPO_FRAME #BASE,POINT2[] " ",TQ_STATE FALSE}
DECL LDAT LCPDAT4={VEL 2.0,ACC 100.0,APO_DIST 10.0,APO_FAC 50.0,AXIS_VEL 100.0,AXIS_ACC 100.0,ORI_TYP #VAR,CIRC_TYP #BASE,JERK_FAC 50.0,GEAR_JERK 50.0,EXAX_IGN 0}
DECL E6POS XP5={X 57.6877289,Y -480.831787,Z 603.130127,A -118.843903,B 79.8543396,C -120.822701,S 18,T 35,E1 0.0,E2 0.0,E3 0.0,E4 0.0,E5 0.0,E6 0.0}
DECL FDAT FP5={TOOL_NO 3,BASE_NO 3,IPO_FRAME #BASE,POINT2[] " ",TQ_STATE FALSE}
DECL LDAT LCPDAT5={VEL 2.0,ACC 90.0,APO_DIST 10.0,APO_FAC 50.0,AXIS_VEL 100.0,AXIS_ACC 100.0,ORI_TYP #VAR,CIRC_TYP #BASE,JERK_FAC 50.0,GEAR_JERK 50.0,EXAX_IGN 0}
DECL E6POS XP7={X 684.034424,Y -664.895325,Z 365.229309,A -22.2569199,B 35.8561401,C -8.6238451,S 18,T 35,E1 0.0,E2 0.0,E3 0.0,E4 0.0,E5 0.0,E6 0.0}
DECL FDAT FP7={TOOL_NO 3,BASE_NO 3,IPO_FRAME #BASE,POINT2[] " ",TQ_STATE FALSE}
DECL LDAT LCPDAT7={VEL 2.0,ACC 100.0,APO_DIST 0.0,APO_FAC 50.0,AXIS_VEL 100.0,AXIS_ACC 100.0,ORI_TYP #VAR,CIRC_TYP #BASE,JERK_FAC 50.0,GEAR_JERK 50.0,EXAX_IGN 0}
DECL E6POS XP8={X 687.160217,Y -664.176697,Z 347.525391,A -22.0968399,B 35.009449,C -8.33810997,S 18,T 35,E1 0.0,E2 0.0,E3 0.0,E4 0.0,E5 0.0,E6 0.0}
DECL FDAT FP8={TOOL_NO 3,BASE_NO 3,IPO_FRAME #BASE,POINT2[] " ",TQ_STATE FALSE}
DECL LDAT LCPDAT8={VEL 2.0,ACC 100.0,APO_DIST 10.0,APO_FAC 50.0,AXIS_VEL 100.0,AXIS_ACC 100.0,ORI_TYP #VAR,CIRC_TYP #BASE,JERK_FAC 50.0,GEAR_JERK 50.0,EXAX_IGN 0}
DECL PDAT PPDAT3={VEL 100.0,ACC 100.0,APO_DIST 100.0,APO_MODE #CDIS,GEAR_JERK 50.0}
DECL PDAT PPDAT4={VEL 100.0,ACC 100.0,APO_DIST 100.0,GEAR_JERK 50.0}
DECL E6POS XP9={X 622.583984,Y -967.26239,Z 1277.27197,A 77.9929962,B -83.6166,C 13.7835302,S 22,T 19,E1 0.0,E2 0.0,E3 0.0,E4 0.0,E5 0.0,E6 0.0}
DECL FDAT FP9={TOOL_NO 3,BASE_NO 3,IPO_FRAME #BASE,POINT2[] " ",TQ_STATE FALSE}
DECL LDAT LCPDAT9={VEL 2.0,ACC 100.0,APO_DIST 10.0,APO_FAC 50.0,AXIS_VEL 100.0,AXIS_ACC 100.0,ORI_TYP #VAR,CIRC_TYP #BASE,JERK_FAC 50.0,GEAR_JERK 50.0,EXAX_IGN 0}
DECL E6POS XP10={X 584.033997,Y -970.713623,Z 1294.93103,A 127.757797,B -84.1197433,C -35.4890289,S 22,T 19,E1 0.0,E2 0.0,E3 0.0,E4 0.0,E5 0.0,E6 0.0}
DECL FDAT FP10={TOOL_NO 3,BASE_NO 3,IPO_FRAME #BASE,POINT2[] " ",TQ_STATE FALSE}
DECL LDAT LCPDAT10={VEL 2.0,ACC 100.0,APO_DIST 0.0,APO_FAC 50.0,AXIS_VEL 100.0,AXIS_ACC 100.0,ORI_TYP #VAR,CIRC_TYP #BASE,JERK_FAC 50.0,GEAR_JERK 50.0,EXAX_IGN 0}
DECL LDAT LCPDAT11={VEL 2.0,ACC 100.0,APO_DIST 30.0,APO_FAC 50.0,AXIS_VEL 100.0,AXIS_ACC 100.0,ORI_TYP #VAR,CIRC_TYP #BASE,JERK_FAC 50.0,GEAR_JERK 50.0,EXAX_IGN 0}
DECL SPOT_SUGG_T LAST_SPOT={GUN[] "2                       ",RETR_CMD[] "#CLO                    ",CHOISE[] "#FIRST                  ",CLO_TM[] "1                       ",PGNO1[] "186                     ",PRESS1[] "0                       ",PGNO2[] "1                       ",PRESS2[] "0                       ",SPOT_PARAMS[] "NORMAL                  "}
DECL E6POS XP13={X 1734.21204,Y -1867.81604,Z 844.310181,A 176.924194,B -49.5563011,C -94.5412521,S 18,T 11,E1 0.0,E2 0.0,E3 0.0,E4 0.0,E5 0.0,E6 0.0}
DECL FDAT FP13={TOOL_NO 3,BASE_NO 3,IPO_FRAME #BASE,POINT2[] " ",TQ_STATE FALSE}
DECL PDAT PPDAT10={VEL 100.0,ACC 80.0,APO_DIST 100.0,APO_MODE #CDIS,GEAR_JERK 50.0}
DECL PDAT PP_OLP7={VEL 100.0,ACC 100.0,APO_DIST 0.0}
DECL E6POS Xl007={X 1644.52502,Y -2192.26294,Z 368.696686,A 170.023499,B -52.7817612,C -87.1773682,S 18,T 3,E1 0.0,E2 0.0,E3 0.0,E4 0.0,E5 0.0,E6 0.0}
DECL FDAT Fl007={TOOL_NO 3,BASE_NO 3,IPO_FRAME #BASE,POINT2[] " "}
DECL PDAT PP_OLP8={VEL 100.0,ACC 100.0,APO_DIST 50.0,APO_MODE #CDIS}
DECL E6POS Xl008={X 745.877075,Y -1613.48499,Z 78.2501373,A -16.3194294,B 12.0206604,C -22.6783009,S 18,T 3,E1 0.0,E2 0.0,E3 0.0,E4 0.0,E5 0.0,E6 0.0}
DECL FDAT Fl008={TOOL_NO 3,BASE_NO 3,IPO_FRAME #BASE,POINT2[] " "}
DECL LDAT LL_OLP65={VEL 2.0,ACC 100.0,APO_DIST 10.0,APO_FAC 0.0,ORI_TYP #VAR,CIRC_TYP #BASE,JERK_FAC 50.0}
DECL E6POS Xl042={X 120.267197,Y -792.371704,Z 628.356201,A -114.714401,B 75.1284332,C -117.9123,S 18,T 35,E1 0.0,E2 0.0,E3 0.0,E4 0.0,E5 0.0,E6 0.0}
DECL FDAT Fl042={TOOL_NO 3,BASE_NO 3,IPO_FRAME #BASE,POINT2[] " "}
DECL E6POS XSWP_60_7345={X 142.049606,Y -899.13092,Z 603.691528,A -111.239601,B 76.1861877,C -116.340202,S 18,T 35,E1 0.0,E2 0.0,E3 0.0,E4 0.0,E5 0.0,E6 0.0}
DECL FDAT FSWP_60_7345={TOOL_NO 3,BASE_NO 3,IPO_FRAME #BASE,POINT2[] " "}
DECL E6POS XSWP_60_7897={X 107.674698,Y -641.697876,Z 600.476318,A -108.5028,B 80.4464569,C -108.3703,S 18,T 35,E1 0.0,E2 0.0,E3 0.0,E4 0.0,E5 0.0,E6 0.0}
DECL FDAT FSWP_60_7897={TOOL_NO 3,BASE_NO 3,IPO_FRAME #BASE,POINT2[] " "}
DECL E6POS XSWP_60_7311={X 92.3450699,Y -351.334198,Z 601.31073,A -131.179901,B 80.0362778,C -134.014496,S 18,T 35,E1 0.0,E2 0.0,E3 0.0,E4 0.0,E5 0.0,E6 0.0}
DECL FDAT FSWP_60_7311={TOOL_NO 3,BASE_NO 3,IPO_FRAME #BASE,POINT2[] " "}
DECL LDAT LCPDAT13={VEL 2.0,ACC 100.0,APO_DIST 100.0,APO_FAC 50.0,AXIS_VEL 100.0,AXIS_ACC 100.0,ORI_TYP #VAR,CIRC_TYP #BASE,JERK_FAC 50.0,GEAR_JERK 50.0,EXAX_IGN 0}
DECL LDAT LCPDAT14={VEL 2.0,ACC 100.0,APO_DIST 100.0,APO_FAC 50.0,AXIS_VEL 100.0,AXIS_ACC 100.0,ORI_TYP #VAR,CIRC_TYP #BASE,JERK_FAC 50.0,GEAR_JERK 50.0,EXAX_IGN 0}
DECL LDAT LCPDAT0={VEL 2.0,ACC 90.0,APO_DIST 5.0,APO_FAC 50.0,AXIS_VEL 100.0,AXIS_ACC 100.0,ORI_TYP #VAR,CIRC_TYP #BASE,JERK_FAC 50.0,GEAR_JERK 50.0,EXAX_IGN 0}
DECL E6POS XP0={X 1113.95496,Y -991.188293,Z 14.3488798,A 179.752701,B -16.1354008,C -89.9455795,S 18,T 43,E1 0.0,E2 0.0,E3 0.0,E4 0.0,E5 0.0,E6 0.0}
DECL FDAT FP0={TOOL_NO 3,BASE_NO 3,IPO_FRAME #BASE,POINT2[] " ",TQ_STATE FALSE}
DECL LDAT LCPDAT15={VEL 2.0,ACC 100.0,APO_DIST 5.0,APO_FAC 50.0,AXIS_VEL 100.0,AXIS_ACC 100.0,ORI_TYP #VAR,CIRC_TYP #BASE,JERK_FAC 50.0,GEAR_JERK 50.0,EXAX_IGN 0}
DECL E6POS XP14={X 1106.151,Y -1003.31702,Z 67.7898407,A 179.753098,B -16.1340904,C -89.9462967,S 18,T 43,E1 0.0,E2 0.0,E3 0.0,E4 0.0,E5 0.0,E6 0.0}
DECL FDAT FP14={TOOL_NO 3,BASE_NO 3,IPO_FRAME #BASE,POINT2[] " ",TQ_STATE FALSE}
DECL LDAT LCPDAT16={VEL 2.0,ACC 100.0,APO_DIST 100.0,APO_FAC 50.0,AXIS_VEL 100.0,AXIS_ACC 100.0,ORI_TYP #VAR,CIRC_TYP #BASE,JERK_FAC 50.0,GEAR_JERK 50.0,EXAX_IGN 0}
DECL E6POS XSWP_61_7027={X 1091.26697,Y -1014.38599,Z 62.79179,A 179.752899,B -16.1340504,C -89.9468307,S 22,T 19,E1 0.0,E2 0.0,E3 0.0,E4 0.0,E5 0.0,E6 0.0}
DECL FDAT FSWP_61_7027={TOOL_NO 3,BASE_NO 3,IPO_FRAME #BASE,POINT2[] " ",TQ_STATE FALSE}
DECL LDAT LCPDAT17={VEL 2.0,ACC 100.0,APO_DIST 100.0,APO_FAC 50.0,AXIS_VEL 100.0,AXIS_ACC 100.0,ORI_TYP #VAR,CIRC_TYP #BASE,JERK_FAC 50.0,GEAR_JERK 50.0,EXAX_IGN 0}
DECL E6POS XSWP_61_7029={X 1176.19299,Y -1021.13898,Z 95.2776031,A 179.752304,B -16.1331501,C -89.9456406,S 18,T 43,E1 0.0,E2 0.0,E3 0.0,E4 0.0,E5 0.0,E6 0.0}
DECL FDAT FSWP_61_7029={TOOL_NO 3,BASE_NO 3,IPO_FRAME #BASE,POINT2[] " ",TQ_STATE FALSE}
DECL E6POS XSWP_61_7031={X 1228.125,Y -1021.565,Z 105.6548,A 179.7388,B -30.3301392,C -89.944603,S 18,T 43,E1 0.0,E2 0.0,E3 0.0,E4 0.0,E5 0.0,E6 0.0}
DECL FDAT FSWP_61_7031={TOOL_NO 3,BASE_NO 3,IPO_FRAME #BASE,POINT2[] " ",TQ_STATE FALSE}
DECL E6POS XP15={X 1282.54199,Y -1002.97803,Z 55.04533,A 179.737793,B -30.3313904,C -89.9422989,S 22,T 19,E1 0.0,E2 0.0,E3 0.0,E4 0.0,E5 0.0,E6 0.0}
DECL FDAT FP15={TOOL_NO 3,BASE_NO 3,IPO_FRAME #BASE,POINT2[] " ",TQ_STATE FALSE}
DECL LDAT LCPDAT21={VEL 2.0,ACC 100.0,APO_DIST 100.0,APO_FAC 50.0,AXIS_VEL 100.0,AXIS_ACC 100.0,ORI_TYP #VAR,CIRC_TYP #BASE,JERK_FAC 50.0,GEAR_JERK 50.0,EXAX_IGN 0}
DECL LDAT LCPDAT22={VEL 2.0,ACC 100.0,APO_DIST 5.0,APO_FAC 50.0,AXIS_VEL 100.0,AXIS_ACC 100.0,ORI_TYP #VAR,CIRC_TYP #BASE,JERK_FAC 50.0,GEAR_JERK 50.0,EXAX_IGN 0}
DECL E6POS Xl013={X 983.371399,Y -1478.85498,Z 590.276611,A 179.957199,B -45.9995995,C -90.0003128,S 18,T 43,E1 0.0,E2 0.0,E3 0.0,E4 0.0,E5 0.0,E6 0.0}
DECL FDAT Fl013={TOOL_NO 3,BASE_NO 3,IPO_FRAME #BASE,POINT2[] " "}
DECL E6POS Xl009={X 1304.05298,Y -1270.36804,Z -0.0250963103,A 179.959503,B -16.0019207,C -90.0033722,S 22,T 19,E1 0.0,E2 0.0,E3 0.0,E4 0.0,E5 0.0,E6 0.0}
DECL FDAT Fl009={TOOL_NO 3,BASE_NO 3,IPO_FRAME #BASE,POINT2[] " "}
DECL LDAT LCPDAT23={VEL 2.0,ACC 100.0,APO_DIST 30.0,APO_FAC 50.0,AXIS_VEL 100.0,AXIS_ACC 100.0,ORI_TYP #VAR,CIRC_TYP #BASE,JERK_FAC 50.0,GEAR_JERK 50.0,EXAX_IGN 0}
DECL LDAT LCPDAT24={VEL 2.0,ACC 100.0,APO_DIST 30.0,APO_FAC 50.0,AXIS_VEL 100.0,AXIS_ACC 100.0,ORI_TYP #VAR,CIRC_TYP #BASE,JERK_FAC 50.0,GEAR_JERK 50.0,EXAX_IGN 0}
DECL E6POS XP16={X 1384.60303,Y -1894.59204,Z 1393.06104,A -86.6525192,B -54.8740196,C 168.649399,S 22,T 19,E1 0.0,E2 0.0,E3 0.0,E4 0.0,E5 0.0,E6 0.0}
DECL FDAT FP16={TOOL_NO 3,BASE_NO 3,IPO_FRAME #BASE,POINT2[] " ",TQ_STATE FALSE}
DECL PDAT PPDAT17={VEL 100.0,ACC 100.0,APO_DIST 100.0,APO_MODE #CDIS,GEAR_JERK 50.0}
DECL LDAT LCPDAT25={VEL 2.0,ACC 100.0,APO_DIST 150.0,APO_FAC 50.0,AXIS_VEL 100.0,AXIS_ACC 100.0,ORI_TYP #VAR,CIRC_TYP #BASE,JERK_FAC 50.0,GEAR_JERK 50.0,EXAX_IGN 0}
ENDDAT
